// TIA Portal V20 export
TYPE "LER_typeWeightCheckTrackingData"
// stored: Access Published
   STRUCT
      finished { ExternalWritable := 'False'} : Bool;
      result { ExternalWritable := 'False'} : Bool;
      data { ExternalWritable := 'False'} : Real;
   END_STRUCT;
END_TYPE
